FUNCTION_BLOCK FB_TestCompositeService EXTENDS FB_CompositeServiceBase
VAR_INPUT
	DependencyOne : UDINT;
	DependencyTwo : UDINT;
	DependencyCount : UINT;
	ExecuteResult : E_PackMLHookResult := E_PackMLHookResult.Busy;
END_VAR

M_UpdateCompositeService();

METHOD PROTECTED H_DeclareServices
IF DependencyCount >= 1 THEN M_AddDependency(ServiceId := DependencyOne); END_IF
IF DependencyCount >= 2 THEN M_AddDependency(ServiceId := DependencyTwo); END_IF
END_METHOD

METHOD PROTECTED H_OnCompositeExecute : E_PackMLHookResult
VAR_INPUT bFirstScan : BOOL; END_VAR
H_OnCompositeExecute := ExecuteResult;
END_METHOD

METHOD PUBLIC M_TestAddDependencyOutsideDefinition : BOOL
VAR_INPUT ServiceIdValue : UDINT; END_VAR
M_TestAddDependencyOutsideDefinition := M_AddDependency(ServiceId := ServiceIdValue);
END_METHOD

METHOD PUBLIC M_TestFailSequence
VAR_INPUT FailedServiceId : UDINT; END_VAR
M_FailSequence(ErrorCode := E_CompositeServiceErrorCode.None, FailedServiceId := FailedServiceId, SourceErrorId := 0, Message := 'Test failure');
END_METHOD

END_FUNCTION_BLOCK

(* stored: Version 1.1.0.1, ProductVersion 3.1.4026.18
   POU FB_TestCompositeService: Id {91fb4d75-56fb-466a-af1d-b34d5ec37424}, SpecialFunc None
   Method H_DeclareServices: Id {4423480a-d1f8-42b0-81cc-e63dc5ef7f72}
   Method H_OnCompositeExecute: Id {06a08594-9169-4684-8f5c-624b9103f18e}
   Method M_TestAddDependencyOutsideDefinition: Id {a45587ff-63a7-4edc-898f-692d5db7da6e}
   Method M_TestFailSequence: Id {326eb050-a229-4490-b1d7-8979049883a9} *)
